FUNCTION_BLOCK Forgetting_Factor
VAR_INPUT
	r_forgetFactor : REAL;
	r_inputValue : REAL;
END_VAR
VAR_OUTPUT
	r_meanValueForget_k : REAL;
END_VAR
VAR
	r_meanValueForget_k1 : REAL;
END_VAR

r_meanValueForget_k := r_meanValueForget_k1*r_forgetFactor + (1-r_forgetFactor)*r_inputValue;
r_meanValueForget_k1 := r_meanValueForget_k;

END_FUNCTION_BLOCK

(* stored: Version 1.1.0.1, ProductVersion 3.1.4022.12
   POU Forgetting_Factor: Id {d1cc2f46-0d79-4925-9e9c-0c799b6d90af}, SpecialFunc None *)
